TYPE M3GotoProcedureStatuses :
STRUCT
	///Is the M3GotoProcedure in a busy state?
	busyStatus: BusyStatus;
	///Is the M3GotoProcedure in a healthy state?
	healthStatus: HealthStatus;
END_STRUCT
END_TYPE

(* stored: Version 1.1.0.1, ProductVersion 3.1.4019.2
   DUT M3GotoProcedureStatuses: Id {e37632e8-e2ec-46e7-842e-099267826865} *)
